PROGRAM PRG_TestsAside
VAR
	
END_VAR

END_PROGRAM

(* stored: Version 1.1.0.1
   POU PRG_TestsAside: Id {fd7a18a6-93f4-4922-8663-21835afdd83e}, SpecialFunc None *)
